VAR_GLOBAL

	fbAct1:FB_ActionneurSimple;	//Act1 corresponds to holding the object
	
	xModeStepForStep :BOOL;
	xNextStep : BOOL;
	
	//pour FB_gestion du mode
	fbMMA:FB_MMA;
	fbCycleAuto:FB_CycleAuto;
	fbCycleInit : FB_CycleInit;
	fbCycleMan : FB_CycleMan;
	
	stParam:ST_Param;
	fbBtn:FB_Btn;
	stIO:ST_IO;
	
	//Tachymetre moteur
	//fbMotor : FB_RegulMoteur;
	fbMotorX : FB_Moteur;
	fbMotorY : FB_Moteur;
	fbMotorZ : FB_Moteur;
	

	 
END_VAR

(* stored: Version 1.1.0.1, ProductVersion 3.1.4020.12
   GVL GVL: Id {29e74ae1-1e66-43a7-ba4b-1961dad16adc} *)
